FUNCTION_BLOCK FB_PickAndPlace EXTENDS FB_Module
(* 
ESTACIÓN DE CARGA - Manual de usuario #31/27

La alimentación de material descrita en el punto anterior realiza el suministro 
de tapas que posteriormente serán montadas en el conjunto preparado en 
el palet. Sin embargo, tras esta fase resulta necesario realizar la carga de 
la tapa sobre el plato divisor. 
Para ello se ha dispuesto el manipulador 
de la imagen, compuesto por un cilindro 
rotolineal, encargado de realizar la elevación 
y posterior giro de un brazo con una pinza 
de dos dedos de apertura paralela. El giro 
de 180º realizado por este elemento, sitúa 
la pinza sobre el punto exacto de descarga 
de la tapa en la primera estación del plato 
divisor.

ESTACIÓN DE INSERCIÓN TAPA - Manual de usuario #33/29

Al igual que sucedía en la estación de inserción 
de eje, la última de las estaciones está encargada 
del montaje de la tapa sobre el conjunto retenido 
en la cinta transportadora.

Como puede observarse en la imagen, el 
manipulador previsto para realizar esta tarea 
presenta idénticas características que el utilizado 
para depositar la tapa sobre el plato divisor. 
Dispone de una pinza de apertura paralela para 
sujetar la tapa, que es elevada y desplazada 
realizando un giro hasta el punto de descarga 
mediante un actuador neumático rotolineal.

*)
VAR_INPUT
	Mover: BOOL := TRUE; // TODO HAY QUE CARGAR O DESCARGAR EN FUNCIÓN DEL RESTO DE LA MÁQUINA Y LAS CONSIGNAS DEL PANEL
END_VAR
VAR_OUTPUT
END_VAR
VAR
	(* Controlador  específico *)
	fbController: FB_PickAndPlace_SFC;

	(* Temporizadores específicos *)
	TPIN: TIME := T#1S;	

	(* Sensores específicos *)
	h0 AT %I*: BOOL; (* Final de carrera horizontal retraida *)
	h1 AT %I*: BOOL; (* Final de carrera horizontal extendido *)
	v1 AT %I*: BOOL; (*Final de carrera vertical abajo*)
	v0 AT %I*: BOOL; (*Final de carrera vertical arriba*)

	(* Actuadores específicos *)
	HOR AT %Q*: BOOL; (* Actuador de extension de brazo horizontal *)
	VER AT %Q*: BOOL; (* Actuador de movimiento vertical de brazo*)
	PIN AT %Q*: BOOL; (*Actuador de pinza de brazo*)
END_VAR

METHOD ModuleControlFlow : BOOL
fbController(
	TPIN 	:= TPIN,
	
	ctInp 	:= ctInp, 
	Mover	:= Mover,
	h0 		:= h0,
	h1 		:= h1,
	v0 		:= v0,
	v1 		:= v1,
	
	ctOut 	=> ctOut);
END_METHOD

METHOD ModulePerformActions : BOOL
VAR_INPUT
END_VAR
// el brazo está en condiciones iniciales h0 y v0
ctOut.IC := h0 AND v0; 

// si no eestamos en modo manual, actualizar los actuadores con el estado del controlador
IF NOT ctInp.Manual THEN
	HOR := fbController.HOR;
	VER := fbController.VER;
	PIN := fbController.PIN;
END_IF
END_METHOD

END_FUNCTION_BLOCK

(* stored: Version 1.1.0.1, ProductVersion 3.1.4024.11
   POU FB_PickAndPlace: Id {0acadc22-7b10-494f-8323-7cb38d3e0455}, SpecialFunc None
   Method ModuleControlFlow: Id {ad50b7d3-ffb1-4d5e-9f1d-9c4b9b9b584c}
   Method ModulePerformActions: Id {e3820e39-c043-40cb-babf-d57ef6c637b0} *)
